ABB RobotStudio station: Proyecto_Robotica.rsstn

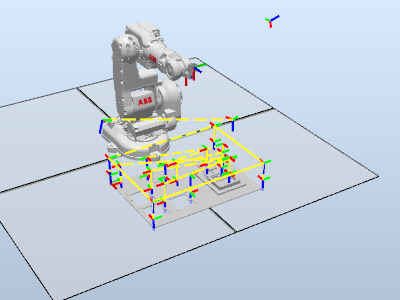
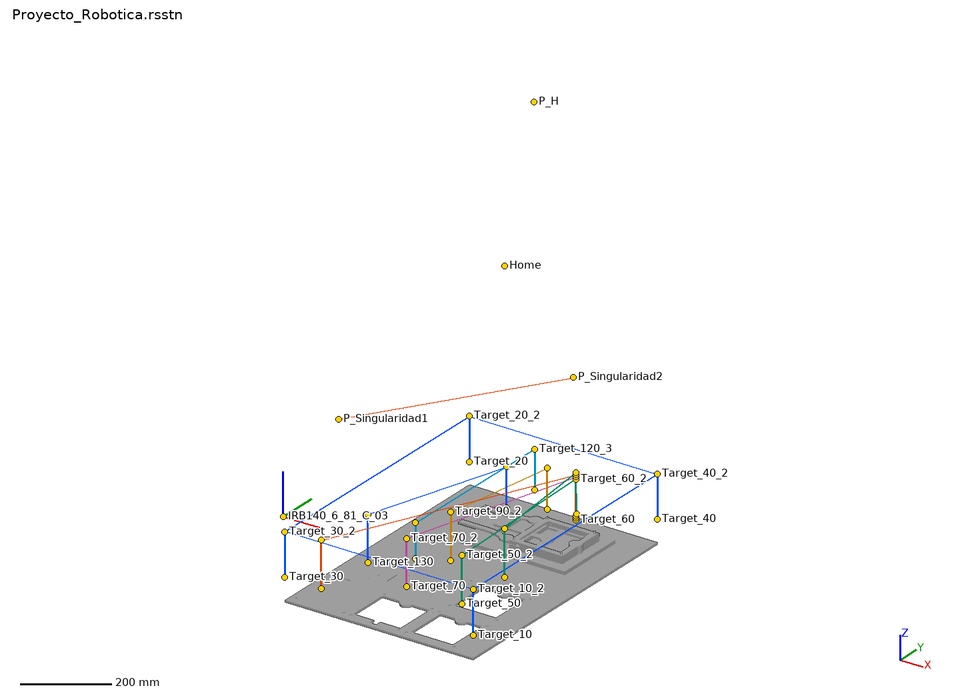
[picture v1: parts stored in the station drawn from their meshes, with robot base, taught points and paths (robot models come from the ABB library and are not in the file)]
Station Proyecto_Robotica (saved by RobotStudio 22.2.10013.1)
Controller Controlador14
  mechanical unit ROB_1: IRB140_6_81_C_03, 6 joints, base frame (0, 0, 0) mm
Layout (positions relative to the parent item):
  - IRB140_6_81_C_03 [mechanism, from Robots\IRB140_6_81_C_G_03.rslib] at (0, 0, 0) mm; joint values [0, 0, 0, 0, 0, 0] (rad or m)
  - P_Tool_v_v2 [mechanism, from Libraries\P_Tool_v_v2.rslib] at (515, 0, 712) mm, rotated rx 0 ry 90 rz 0 deg
  - Base [part] at (745.94, -344.6, 0) mm, rotated rx 0 ry 0 rz -90 deg, size 700 x 500 x 39 mm
  - P1 [part] at (687.15, -190.77, 0) mm, rotated rx 0 ry 0 rz -90 deg, size 142.7 x 140 x 5 mm
  - P1_2 [part] at (649.5, 131, 14) mm, rotated rx 0 ry 0 rz 180 deg, size 142.7 x 140 x 5 mm
  - P2 [part] at (687.15, -27.96, 0) mm, rotated rx 0 ry 0 rz -90 deg, size 142.7 x 140 x 5 mm
  - P4 [part] at (539.54, -189.7, 0) mm, rotated rx 0 ry 0 rz -90 deg, size 142.7 x 140 x 5 mm
  - P4_2 [part] at (649.5, 131, 19) mm, rotated rx 0 ry 0 rz 180 deg, size 142.7 x 140 x 5 mm
  - P3 [part] at (535, -27.36, 0) mm, rotated rx 0 ry 0 rz -90 deg, size 152.7 x 122 x 5 mm
  - P3_2 [part] at (573.73, 140.01, 19) mm, rotated rx 0 ry 0 rz 180 deg, size 152.7 x 122 x 5 mm
  - P5 [part] at (439.32, -63.45, 0) mm, rotated rx 0 ry 0 rz -90 deg, size 85.4 x 163.2 x 5 mm
  - P5_2 [part] at (523.37, 269.08, 24) mm, rotated rx 0 ry 0 rz -90 deg, size 85.4 x 163.2 x 5 mm
  - P7 [part] at (392.94, -216.23, 0) mm, rotated rx 0 ry 0 rz -90 deg, size 116 x 140 x 5 mm
  - P6 [part] at (346.69, -119.92, 0) mm, rotated rx 0 ry 0 rz -90 deg, size 163.2 x 85.4 x 5 mm
  - P6_2 [part] at (523.33, 132.93, 24) mm, rotated rx 0 ry 0 rz 180 deg, size 163.2 x 85.4 x 5 mm
  - P7_2 [part] at (536.11, 271.06, 24) mm, size 116 x 140 x 5 mm
  - P2_2 [part] at (649.5, 131, 29) mm, rotated rx 0 ry 0 rz 180 deg, size 142.7 x 140 x 5 mm
Attachment: P_Tool_v_v2 is attached to IRB140_6_81_C_03 / Link6
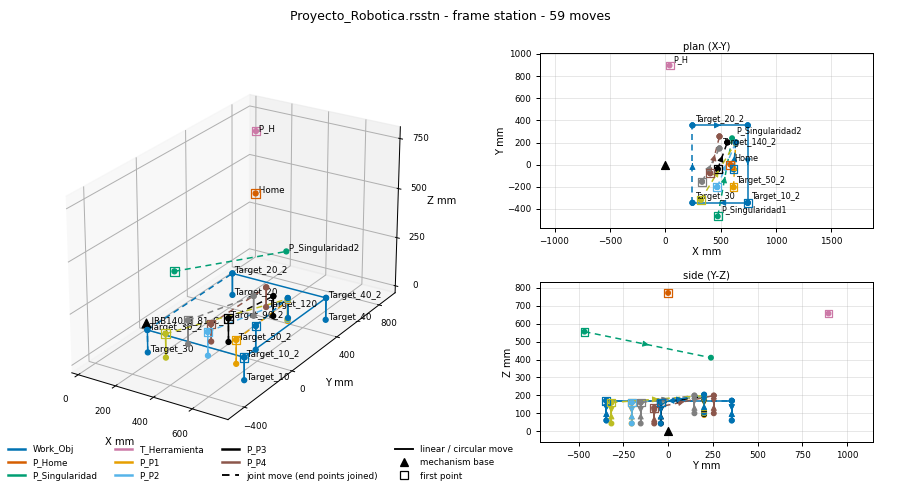
[picture p0: tool path of Proyecto_Robotica.rsstn in frame station, 59 of 59 moves have a stored position in this frame; points joined in program order, loops and branches not executed]
Targets, tools, work objects and paths stored in the station, written as RAPID:
! task T_ROB1
MODULE CalibData
  PERS tooldata TCP_P_Tool_v_v2:=[TRUE,[[-60,0,74],[1,0,0,0]],[1,[0,0,1],[1,0,0,0],0,0,0]];
  TASK PERS wobjdata P_Wob_1:=[FALSE,TRUE,"",[[245.944,-344.596,5],[1,0,0,0]],[[0,0,0],[1,0,0,0]]];
ENDMODULE

! task T_ROB1
MODULE Module1
  CONST robtarget Target_10:=[[500,0,55],[0,0,1,0],[0,0,0,0],[9E+09,9E+09,9E+09,9E+09,9E+09,9E+09]];
  CONST robtarget Target_20:=[[0,700,55],[0,0,1,0],[0,0,0,0],[9E+09,9E+09,9E+09,9E+09,9E+09,9E+09]];
  CONST robtarget Target_30:=[[0,0,55],[0,0,1,0],[-1,0,-1,0],[9E+09,9E+09,9E+09,9E+09,9E+09,9E+09]];
  CONST robtarget Target_40:=[[500,700,55],[0,0,1,0],[0,0,0,0],[9E+09,9E+09,9E+09,9E+09,9E+09,9E+09]];
  CONST robtarget Target_10_2:=[[500,0,165],[0,0,1,0],[0,0,0,0],[9E+09,9E+09,9E+09,9E+09,9E+09,9E+09]];
  CONST robtarget Target_20_2:=[[0,700,165],[0,0,1,0],[0,0,0,0],[9E+09,9E+09,9E+09,9E+09,9E+09,9E+09]];
  CONST robtarget Target_30_2:=[[0,0,165],[0,0,1,0],[-1,0,-1,0],[9E+09,9E+09,9E+09,9E+09,9E+09,9E+09]];
  CONST robtarget Target_40_2:=[[500,700,165],[0,0,1,0],[0,0,0,0],[9E+09,9E+09,9E+09,9E+09,9E+09,9E+09]];
  CONST robtarget Home:=[[343.056,344.596,767],[0.707106781,0,0.707106781,0],[0,0,0,0],[9E+09,9E+09,9E+09,9E+09,9E+09,9E+09]];
  CONST robtarget P_Singularidad1:=[[228.915,-122.332,550.806],[0.353553391,0.35355339,0.853553391,-0.146446609],[0,0,0,0],[9E+09,9E+09,9E+09,9E+09,9E+09,9E+09]];
  CONST robtarget P_Singularidad2:=[[357.952,583.679,405.477],[0,-0.173648177,0.984807753,0],[0,0,0,0],[9E+09,9E+09,9E+09,9E+09,9E+09,9E+09]];
  CONST robtarget P_H:=[[-206.12,1240.192,652.05],[0.560985528,-0.430459334,0.430459334,0.560985527],[0,0,0,0],[9E+09,9E+09,9E+09,9E+09,9E+09,9E+09]];
  CONST robtarget Target_50:=[[371.202,140.828,38],[0,-0.707106781,0.707106781,0],[-1,0,-2,0],[9E+09,9E+09,9E+09,9E+09,9E+09,9E+09]];
  CONST robtarget Target_50_2:=[[371.202,140.828,155],[0,-0.707106781,0.707106781,0],[-1,0,-2,0],[9E+09,9E+09,9E+09,9E+09,9E+09,9E+09]];
  CONST robtarget Target_60:=[[390.556,545.596,85],[0,0,1,0],[0,0,0,0],[9E+09,9E+09,9E+09,9E+09,9E+09,9E+09]];
  CONST robtarget Target_60_2:=[[390.556,545.596,184],[0,0,1,0],[0,0,0,0],[9E+09,9E+09,9E+09,9E+09,9E+09,9E+09]];
  CONST robtarget Target_70:=[[223.599,141.895,38],[0,-0.707106781,0.707106781,0],[-1,0,-2,0],[9E+09,9E+09,9E+09,9E+09,9E+09,9E+09]];
  CONST robtarget Target_80:=[[390.556,545.596,90],[0,0,1,0],[0,0,0,0],[9E+09,9E+09,9E+09,9E+09,9E+09,9E+09]];
  CONST robtarget Target_70_2:=[[223.599,141.895,155],[0,-0.707106781,0.707106781,0],[-1,0,-2,0],[9E+09,9E+09,9E+09,9E+09,9E+09,9E+09]];
  CONST robtarget Target_80_2:=[[390.556,545.596,189],[0,0,1,0],[0,0,0,0],[9E+09,9E+09,9E+09,9E+09,9E+09,9E+09]];
  CONST robtarget Target_90:=[[228.058,304.237,38],[0,-0.707106781,0.707106781,0],[-1,0,-2,0],[9E+09,9E+09,9E+09,9E+09,9E+09,9E+09]];
  CONST robtarget Target_100:=[[314.785,545.604,90],[0,0,1,0],[0,0,0,0],[9E+09,9E+09,9E+09,9E+09,9E+09,9E+09]];
  CONST robtarget Target_90_2:=[[228.058,304.237,155],[0,-0.707106781,0.707106781,0],[-1,0,-2,0],[9E+09,9E+09,9E+09,9E+09,9E+09,9E+09]];
  CONST robtarget Target_100_2:=[[314.785,545.604,189],[0,0,1,0],[0,0,0,0],[9E+09,9E+09,9E+09,9E+09,9E+09,9E+09]];
  CONST robtarget Target_110:=[[160.187,267.153,38],[0,1,0,0],[-1,-2,1,0],[9E+09,9E+09,9E+09,9E+09,9E+09,9E+09]];
  CONST robtarget Target_110_2:=[[160.187,267.153,125],[0,1,0,0],[0,0,0,0],[9E+09,9E+09,9E+09,9E+09,9E+09,9E+09]];
  CONST robtarget Target_130:=[[86.75,191.488,38],[0,1,0,0],[-1,0,1,0],[9E+09,9E+09,9E+09,9E+09,9E+09,9E+09]];
  CONST robtarget Target_130_2:=[[86.75,191.488,155],[0,1,0,0],[0,0,0,0],[9E+09,9E+09,9E+09,9E+09,9E+09,9E+09]];
  CONST robtarget Target_120:=[[244.233,599.681,95],[0,1,0,0],[0,0,-2,0],[9E+09,9E+09,9E+09,9E+09,9E+09,9E+09]];
  CONST robtarget Target_120_3:=[[244.233,599.681,194],[0,1,0,0],[0,0,-2,0],[9E+09,9E+09,9E+09,9E+09,9E+09,9E+09]];
  CONST robtarget Target_140:=[[244.194,491.521,95],[0,-0.707106781,0.707106781,0],[0,0,-1,0],[9E+09,9E+09,9E+09,9E+09,9E+09,9E+09]];
  CONST robtarget Target_140_2:=[[244.194,491.521,194],[0,-0.707106781,0.707106781,0],[0,0,-1,0],[9E+09,9E+09,9E+09,9E+09,9E+09,9E+09]];
  CONST robtarget Target_150:=[[77,28,38],[0,-0.707106781,0.707106781,0],[-1,0,-2,0],[9E+09,9E+09,9E+09,9E+09,9E+09,9E+09]];
  CONST robtarget Target_150_3:=[[77,28,155],[0,-0.707106781,0.707106781,0],[-1,0,-2,0],[9E+09,9E+09,9E+09,9E+09,9E+09,9E+09]];
  CONST robtarget Target_160:=[[390.532,545.66,95],[0,1,0,0],[0,0,-2,0],[9E+09,9E+09,9E+09,9E+09,9E+09,9E+09]];
  CONST robtarget Target_160_2:=[[390.532,545.66,194],[0,1,0,0],[0,0,-2,0],[9E+09,9E+09,9E+09,9E+09,9E+09,9E+09]];
  CONST robtarget Target_170:=[[371.202,303.635,38],[0,0.707106781,0.707106781,0],[0,0,1,0],[9E+09,9E+09,9E+09,9E+09,9E+09,9E+09]];
  CONST robtarget Target_170_2:=[[371.202,303.635,155],[0,0.707106781,0.707106781,0],[0,0,0,0],[9E+09,9E+09,9E+09,9E+09,9E+09,9E+09]];
  CONST robtarget Target_180:=[[392.556,545.596,100],[0,1,0,0],[0,0,-2,0],[9E+09,9E+09,9E+09,9E+09,9E+09,9E+09]];
  CONST robtarget Target_180_2:=[[390.556,545.596,199],[0,1,0,0],[0,0,-2,0],[9E+09,9E+09,9E+09,9E+09,9E+09,9E+09]];
  PROC Work_Obj()
    MoveJ Target_10_2,v150,z10,TCP_P_Tool_v_v2\WObj:=P_Wob_1;
    MoveL Target_10,v150,z10,TCP_P_Tool_v_v2\WObj:=P_Wob_1;
    MoveL Target_10_2,v150,z10,TCP_P_Tool_v_v2\WObj:=P_Wob_1;
    MoveL Target_30_2,v150,z10,TCP_P_Tool_v_v2\WObj:=P_Wob_1;
    MoveL Target_30,v150,z10,TCP_P_Tool_v_v2\WObj:=P_Wob_1;
    MoveJ Target_30_2,v150,z10,TCP_P_Tool_v_v2\WObj:=P_Wob_1;
    MoveJ Target_20_2,v150,z10,TCP_P_Tool_v_v2\WObj:=P_Wob_1;
    MoveL Target_20,v150,z10,TCP_P_Tool_v_v2\WObj:=P_Wob_1;
    MoveL Target_20_2,v150,z10,TCP_P_Tool_v_v2\WObj:=P_Wob_1;
    MoveL Target_40_2,v150,z10,TCP_P_Tool_v_v2\WObj:=P_Wob_1;
    MoveL Target_40,v150,z10,TCP_P_Tool_v_v2\WObj:=P_Wob_1;
    MoveL Target_40_2,v150,z10,TCP_P_Tool_v_v2\WObj:=P_Wob_1;
    MoveL Target_10_2,v150,z10,TCP_P_Tool_v_v2\WObj:=P_Wob_1;
  ENDPROC
  PROC P_Home()
    MoveJ Home,v150,z10,TCP_P_Tool_v_v2\WObj:=P_Wob_1;
  ENDPROC
  PROC P_Singularidad()
    MoveJ P_Singularidad1,v150,z10,TCP_P_Tool_v_v2\WObj:=P_Wob_1;
    MoveJ P_Singularidad2,v150,z10,TCP_P_Tool_v_v2\WObj:=P_Wob_1;
  ENDPROC
  PROC T_Herramienta()
    MoveJ P_H,v150,z10,TCP_P_Tool_v_v2\WObj:=P_Wob_1;
  ENDPROC
  PROC P_P1()
    MoveJ Target_50_2,v150,z10,TCP_P_Tool_v_v2\WObj:=P_Wob_1;
    MoveL Target_50,v150,z10,TCP_P_Tool_v_v2\WObj:=P_Wob_1;
    MoveJ Target_50_2,v150,z10,TCP_P_Tool_v_v2\WObj:=P_Wob_1;
    MoveJ Target_60_2,v150,z10,TCP_P_Tool_v_v2\WObj:=P_Wob_1;
    MoveL Target_60,v150,z10,TCP_P_Tool_v_v2\WObj:=P_Wob_1;
    MoveL Target_60_2,v150,z10,TCP_P_Tool_v_v2\WObj:=P_Wob_1;
  ENDPROC
  PROC P_P2()
    MoveJ Target_70_2,v150,z10,TCP_P_Tool_v_v2\WObj:=P_Wob_1;
    MoveL Target_70,v150,z10,TCP_P_Tool_v_v2\WObj:=P_Wob_1;
    MoveJ Target_70_2,v150,z10,TCP_P_Tool_v_v2\WObj:=P_Wob_1;
    MoveJ Target_80_2,v150,z10,TCP_P_Tool_v_v2\WObj:=P_Wob_1;
    MoveL Target_80,v150,z10,TCP_P_Tool_v_v2\WObj:=P_Wob_1;
    MoveL Target_80_2,v150,z10,TCP_P_Tool_v_v2\WObj:=P_Wob_1;
  ENDPROC
  PROC P_P3()
    MoveJ Target_90_2,v150,z10,TCP_P_Tool_v_v2\WObj:=P_Wob_1;
    MoveL Target_90,v150,z10,TCP_P_Tool_v_v2\WObj:=P_Wob_1;
    MoveJ Target_90_2,v150,z10,TCP_P_Tool_v_v2\WObj:=P_Wob_1;
    MoveJ Target_100_2,v150,z10,TCP_P_Tool_v_v2\WObj:=P_Wob_1;
    MoveL Target_100,v150,z10,TCP_P_Tool_v_v2\WObj:=P_Wob_1;
    MoveL Target_100_2,v150,z10,TCP_P_Tool_v_v2\WObj:=P_Wob_1;
  ENDPROC
  PROC P_P4()
    MoveJ Target_110_2,v150,z10,TCP_P_Tool_v_v2\WObj:=P_Wob_1;
    MoveL Target_110,v150,z10,TCP_P_Tool_v_v2\WObj:=P_Wob_1;
    MoveL Target_110_2,v150,z10,TCP_P_Tool_v_v2\WObj:=P_Wob_1;
    MoveJ Target_120_3,v150,z10,TCP_P_Tool_v_v2\WObj:=P_Wob_1;
    MoveL Target_120,v150,z10,TCP_P_Tool_v_v2\WObj:=P_Wob_1;
    MoveL Target_120_3,v150,z10,TCP_P_Tool_v_v2\WObj:=P_Wob_1;
  ENDPROC
  PROC P_P5()
    MoveJ Target_130_2,v150,z10,TCP_P_Tool_v_v2\WObj:=P_Wob_1;
    MoveL Target_130,v150,z10,TCP_P_Tool_v_v2\WObj:=P_Wob_1;
    MoveL Target_130_2,v150,z10,TCP_P_Tool_v_v2\WObj:=P_Wob_1;
    MoveJ Target_140_2,v150,z10,TCP_P_Tool_v_v2\WObj:=P_Wob_1;
    MoveL Target_140,v150,z10,TCP_P_Tool_v_v2\WObj:=P_Wob_1;
    MoveL Target_140_2,v150,z10,TCP_P_Tool_v_v2\WObj:=P_Wob_1;
  ENDPROC
  PROC P_P6()
    MoveJ Target_150_3,v150,z10,TCP_P_Tool_v_v2\WObj:=P_Wob_1;
    MoveL Target_150,v150,z10,TCP_P_Tool_v_v2\WObj:=P_Wob_1;
    MoveL Target_150_3,v150,z10,TCP_P_Tool_v_v2\WObj:=P_Wob_1;
    MoveJ Target_160_2,v150,z10,TCP_P_Tool_v_v2\WObj:=P_Wob_1;
    MoveL Target_160,v150,z10,TCP_P_Tool_v_v2\WObj:=P_Wob_1;
    MoveL Target_160_2,v150,z10,TCP_P_Tool_v_v2\WObj:=P_Wob_1;
  ENDPROC
  PROC P_P7()
    MoveJ Target_170_2,v150,z10,TCP_P_Tool_v_v2\WObj:=P_Wob_1;
    MoveL Target_170,v150,z10,TCP_P_Tool_v_v2\WObj:=P_Wob_1;
    MoveL Target_170_2,v150,z10,TCP_P_Tool_v_v2\WObj:=P_Wob_1;
    MoveJ Target_180_2,v150,z10,TCP_P_Tool_v_v2\WObj:=P_Wob_1;
    MoveL Target_180,v150,z10,TCP_P_Tool_v_v2\WObj:=P_Wob_1;
    MoveL Target_180_2,v150,z10,TCP_P_Tool_v_v2\WObj:=P_Wob_1;
  ENDPROC
ENDMODULE

